FUNCTION_BLOCK FB_Conveyor

VAR_INPUT
    bStart          : BOOL;
    bStop           : BOOL;
    bReset          : BOOL;
    bEmergencyStop  : BOOL;
END_VAR

VAR_OUTPUT
    stStatus        : ST_ConveyorStatus;
END_VAR

VAR
    rStart : R_TRIG;
    rStop  : R_TRIG;
    rReset : R_TRIG;
END_VAR

rStart(CLK := bStart);
rStop(CLK := bStop);
rReset(CLK := bReset);

// Emergency Stop has the highest priority
IF bEmergencyStop THEN
    stStatus.eState := E_MachineState.Faulted;
END_IF;

// Reset clears the fault
IF rReset.Q THEN
    stStatus.eState := E_MachineState.Stopped;
END_IF;

// Main machine state
CASE stStatus.eState OF

    E_MachineState.Stopped:

        stStatus.bMotorRunning := FALSE;

        IF rStart.Q THEN
            stStatus.eState := E_MachineState.Starting;
        END_IF


    E_MachineState.Starting:

        stStatus.bMotorRunning := TRUE;
        stStatus.eState := E_MachineState.Running;


    E_MachineState.Running:

        stStatus.bMotorRunning := TRUE;

        IF rStop.Q THEN
            stStatus.eState := E_MachineState.Stopping;
        END_IF


    E_MachineState.Stopping:

        stStatus.bMotorRunning := FALSE;
        stStatus.eState := E_MachineState.Stopped;


    E_MachineState.Faulted:

        stStatus.bMotorRunning := FALSE;

END_CASE;

END_FUNCTION_BLOCK

(* stored: Version 1.1.0.1, ProductVersion 3.1.4026.18
   POU FB_Conveyor: Id {cd65f802-7882-40c4-9d72-4194747e95ad}, SpecialFunc None *)
